// TIA Portal V21 export
TYPE "Std_Stazione"
   STRUCT
      IN : Struct
         CodiceProdotto : Int;   // Indica il codice lavorato attualmente dalla stazione
         Portata : Real;   // Indica il flusso prodotto, espresso in metri cubi/litri/bottiglie/etc
      END_STRUCT;
      Prm : Struct
         Partner : Struct
            TipoAssociazione : Byte;   // 0=Completa(Comporta richiesta di associazione e verifica fattibilità del percorso se possibile controlla la chiamata partner) 1 = SoloStato (Verifica solo lo stato della chiamata partner)
         END_STRUCT;
         CadutaChiamata : Struct   // Condizioni di caduta di chiamata verso monte
            DaAnalogicaPer : Struct   // Funzioni dell'analogica
               SogliaMaxi : Byte;   // 0=Disabiliatato 1=Raggiunta 2=NonRaggiunta (ES: Se raggiungo la soglia Massima ed il parametro è impostato ad 1 cade la chiamata)
               SogliaIntMax : Byte;   // 0=Disabiliatato 1=Raggiunta 2=NonRaggiunta (ES: Se non raggiungo la soglia IntMax ed il parametro è impostato a 2 cade la chiamata)
               SogliaIntMin : Byte;   // 0=Disabiliatato 1=Raggiunta 2=NonRaggiunta (ES: Se raggiungo la soglia IntMin ed il parametro è impostato ad 1 cade la chiamata)
               SogliaMini : Byte;   // 0=Disabiliatato 1=Raggiunta 2=NonRaggiunta (ES: Se non raggiungo la soglia Minima ed il parametro è impostato a 2 cade la chiamata)
            END_STRUCT;
         END_STRUCT;
         BypassDestinazione : Bool;   // Se impostato ad 1 la stazione chiama senza tener conto della destinazione quando non c'è nessuna destinazione attiva e se è presente almeno una stazione sorgente attiva
         BypassSorgente : Bool;   // Se impostato ad 1 insieme al "BypassDestinazione" la stazione chiama senza tener conto della destinazione quando non c'è nessuna destinazione attiva e senza tenere conto delle sorgenti
      END_STRUCT;
      Hmi : Struct
         Abilita : Bool;   // Selettore di abilitazione ad HMI
         ByPassConsensoMacchina : Bool;
         Diagnostica : Struct
            "00-Analogica" : Bool;   // 0 - Non in chiamata causa analogica associata
            "01-Paratia" : Bool;   // 1- Non in chiamata causa paratia associata
            "02-Motore" : Bool;   // 2 - Non in chiamata causa motore associato
            "03-Pompa" : Bool;   // 3 - Non in chiamata causa pompa associata
            "04-NessunaStazioneInChiamata" : Bool;   // 4 - Nessuna stazione attiva in chiamata
            "05-StopChiamataDaPLC" : Bool;   // 5 - Chiamata verso monte fermata da PLC
            "06-SelettoreHMIStop" : Bool;   // 6 - Chiamata verso monte fermata da selettore HMI
            "07-MancanzaConsensoMacchina" : Bool;   // 7- Mancanza consenso macchina
            "08-StazionePartnerNonChiama" : Bool;   // 8 - La stazione partner è associata ma non è attualmente in chiamata
            "09-" : Bool;
         END_STRUCT;
      END_STRUCT;
      Allarmi : Struct
         Stato : Struct
            ConflittoMultiDest : Bool;
         END_STRUCT;
         EnWarnHmi : Struct
            ConflittoMultiDest : Bool;
         END_STRUCT;
         WordHMI : Word;
      END_STRUCT;
      Destinazione : Array[0.."K_NumStazione"] of "Std_Stazioni";
      Dati : Struct
         DestAttivaPresente : Bool;   // Inidica che per la presente stazione almeno una destinazione progettata è attiva (Percorso attivo online)
         SorgAttivaPresente : Bool;   // Inidica che per la presente stazione almeno una sorgente progettata è attiva (Percorso attivo online)
         AlmenoUnaSorgenteProgettata : Bool;   // Inidica che per la presente stazione è progettata almeno una sorgente
         AlmenoUnaDestinazioneProgettata : Bool;   // Inidica che per la presente stazione è progettata almeno una destinazione
      END_STRUCT;
      OUT : Struct
         Chiamata : Bool;
      END_STRUCT;
      Rif_Inc : Struct
         K_Analogica : Int;
         K_Paratia : Int;
         K_Motore : Int;
         K_Pompa : Int;
         K_Stazione : Int;
      END_STRUCT;
   END_STRUCT;
END_TYPE
